FUNCTION_BLOCK GroupController
VAR CONSTANT
	MAX_LIGHTS : INT := 50;
END_VAR
VAR_INPUT
END_VAR
VAR_OUTPUT
END_VAR
VAR
	shuttersCloseRequested : BOOL := FALSE;
	shuttersOpenRequested : BOOL := FALSE;
	
	shutterMoveInterval : TP := (PT := T#10S);
	currentShutterNumber : INT := 1;
END_VAR

METHOD PRIVATE getSource : STRING
VAR_INPUT
END_VAR

VAR
END_VAR
getSource := ' - Group controller';
END_METHOD

METHOD PUBLIC groupShutterLoop

VAR_INPUT
	shutters : ARRAY[1..GVL.MAX_SHUTTERS] OF ShutterSwitch;
END_VAR

VAR

END_VAR
IF NOT shuttersCloseRequested THEN
	JMP _ret;
END_IF

shutterMoveInterval(IN:= FALSE);

IF NOT shutterMoveInterval.Q THEN
	GVL.EventLogger.print3(level:= TcEventSeverity.Verbose, str1:='Closing shutter number=', str2:= TO_STRING(currentShutterNumber), str3:=getSource());
	shutterMoveInterval(IN:= TRUE);
	shutters[currentShutterNumber].moveDownMax(requestedExternally:= TRUE);
	currentShutterNumber := currentShutterNumber + 1;
END_IF

IF currentShutterNumber > GVL.MAX_SHUTTERS THEN
	GVL.EventLogger.print3(level:= TcEventSeverity.Verbose, str1:='Closing shutters finished, closed=', str2:= TO_STRING(currentShutterNumber-1), str3:=getSource());
	shuttersCloseRequested := FALSE;
	currentShutterNumber := 1;
END_IF
 
_ret :


IF NOT shuttersOpenRequested THEN
	JMP _ret2;
END_IF

shutterMoveInterval(IN:= FALSE);

IF NOT shutterMoveInterval.Q THEN
	GVL.EventLogger.print3(level:= TcEventSeverity.Verbose, str1:='Opening shutter number=', str2:= TO_STRING(currentShutterNumber), str3:=getSource());
	shutterMoveInterval(IN:= TRUE);
	shutters[currentShutterNumber].moveUpMax(requestedExternally:= TRUE);
	currentShutterNumber := currentShutterNumber + 1;
END_IF

IF currentShutterNumber > GVL.MAX_SHUTTERS THEN
	GVL.EventLogger.print3(level:= TcEventSeverity.Verbose, str1:='Opening shutters finished, closed=', str2:= TO_STRING(currentShutterNumber), str3:=getSource());
	shuttersOpenRequested := FALSE;
	currentShutterNumber := 1;
END_IF

_ret2 :
END_METHOD

METHOD requestLightsOff : BOOL
VAR_INPUT
	lights : ARRAY[1..MAX_LIGHTS] OF LightSwitch;
END_VAR

VAR
	i : INT;
END_VAR
GVL.EventLogger.print3(level:= TcEventSeverity.Info, str1:='Lights OFF requested', str2:= '', str3:=getSource());

FOR i := 1 TO MAX_LIGHTS BY 1 DO
	lights[i].turnOff();
END_FOR
END_METHOD

METHOD requestLightsOnDefault : BOOL
VAR_INPUT
	lights : ARRAY[1..MAX_LIGHTS] OF LightSwitch;
END_VAR

VAR
	i : INT;
END_VAR
GVL.EventLogger.print3(level:= TcEventSeverity.Info, str1:='Lights ON default requested', str2:= '', str3:=getSource());

FOR i := 1 TO MAX_LIGHTS BY 1 DO
	lights[i].turnOnDefault();
END_FOR
END_METHOD

METHOD PUBLIC requestShuttersClose : BOOL
VAR_INPUT
END_VAR
GVL.EventLogger.print3(level:= TcEventSeverity.Info, str1:='Shutters CLOSE requested', str2:= '', str3:=getSource());

shuttersCloseRequested := TRUE;
shuttersOpenRequested := FALSE;
currentShutterNumber := 1;
END_METHOD

METHOD PUBLIC requestShuttersOpen : BOOL
VAR_INPUT
END_VAR
GVL.EventLogger.print3(level:= TcEventSeverity.Info, str1:='Shutters OPEN requested', str2:= '', str3:=getSource());

shuttersOpenRequested := TRUE;
shuttersCloseRequested := FALSE;
currentShutterNumber := 1;
END_METHOD

END_FUNCTION_BLOCK

(* stored: Version 1.1.0.1, ProductVersion 3.1.4024.12
   POU GroupController: Id {9e2dea4c-15e9-4ccb-84f0-bf94eaeca36c}, SpecialFunc None
   Method getSource: Id {fb3e8195-c629-4336-a586-72d85972302e}
   Method groupShutterLoop: Id {902b955c-86fb-4bb2-a5a6-c864a54d98be}
   Method requestLightsOff: Id {985aeeea-4a3c-4846-a7a2-a8f187eeda96}
   Method requestLightsOnDefault: Id {71279285-d9e5-48b2-ac31-d797ca22a13a}
   Method requestShuttersClose: Id {f3fde636-7658-4863-a5d1-01bc94f61d8d}
   Method requestShuttersOpen: Id {a8b16986-9729-40f4-b5dc-f0d2780e881a} *)
